PROGRAM MAIN
VAR
	_Peripherie	: Peripherie;
	
END_VAR

_Peripherie.Run();
_Peripherie.RtcSynchronize(TRUE, '', 60);

END_PROGRAM

(* stored: Version 1.1.0.1
   POU MAIN: Id {5a046460-1c21-44ae-886d-7aad596c85fa}, SpecialFunc None *)
